{attribute addProperty BoxType "EL1262-0000-0002"}
{attribute addProperty Id "StartTimeNextLatchAT %I*UDINT324"}
{attribute addProperty CRC "3938723629"}
{attribute addProperty SizeInBites "32"}
{attribute addProperty SizeInBytes "4"}
TYPE NextSync1Time_EAC4272D :
STRUCT
	{attribute addProperty Name "StartTimeNextLatch"}
	StartTimeNextLatch AT %I* : UDINT;
END_STRUCT
END_TYPE

(* stored: Version 1.2.0.0, ProductVersion 3.1.4024.9
   DUT NextSync1Time_EAC4272D: Id {cfaf05d6-802f-405e-915b-f415c360605f} *)
